Universal Robots PolyScope program: cover corner demo.urp

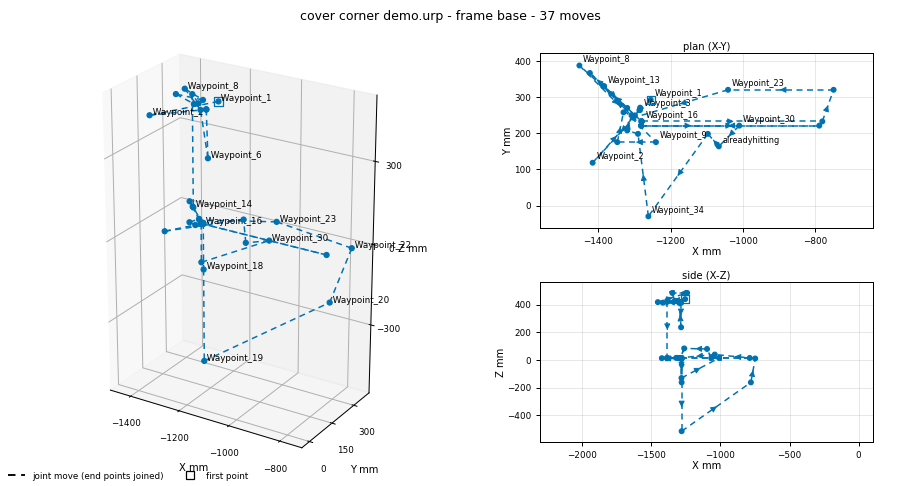
[picture p0: tool path of cover corner demo.urp in frame base, 37 of 37 moves have a stored position in this frame; points joined in program order, loops and branches not executed]
Program cover corner demo (installation=default directory=/programs createdIn=5.21.3 lastSavedIn=5.21.3 robotSerialNumber=20246801938)
Calibrated DH parameters: a=[-0.000071, -0.790281, -0.600694, 0.000061, -0.000039, 0]; d=[0.236272, 604.465945, 132.116513, -736.382239, 0.159268, 0.154005]; alpha=[1.570254, -0.000567, 0.000559, 1.571709, -1.56999, 0]; deltaTheta=[0, -0.409357, 7.293326, -0.600784, -0.000001, -0.000001]
InitVariablesNode
Robot Program (runOnlyOnce=true)
  'right cover corner weld'
  'around then straight'
  MoveJ speed 60 deg/s, acceleration 80 deg/s^2 (useActiveTCP=true optimoveEnabled=false optiMoveSpeed=0.3 optiMoveAcceleration=0.09) feature=Base
    Waypoint Waypoint_1: TCP in base x=-1254.835 y=293.144 z=440.638 mm, rx=-1.1133 ry=-2.919 rz=-0.012 rad; joints [-17.342, -68.282, 77.268, -10.218, 114.462, -0.524] deg; TCP offset x=4.51 y=-328 z=105.73 mm, rx=1.2092 ry=-1.2092 rz=1.2092 rad
  MoveJ speed 60 deg/s, acceleration 80 deg/s^2 (useActiveTCP=true optimoveEnabled=false optiMoveSpeed=0.3 optiMoveAcceleration=0.09) feature=Base
    'around'
    Waypoint Waypoint_2: TCP in base x=-1415.792 y=118.619 z=414.89 mm, rx=-1.1133 ry=-2.919 rz=-0.012 rad; joints [-6.875, -56.934, 61.751, -6.179, 124.925, -0.802] deg
    Waypoint Waypoint_3: TCP in base x=-1285.353 y=264.728 z=415.081 mm, rx=-1.1133 ry=-2.919 rz=-0.012 rad; joints [-15.395, -66.104, 76.117, -11.264, 116.409, -0.572] deg
    Waypoint Waypoint_4: TCP in base x=-1285.353 y=264.728 z=415.081 mm, rx=-0.9669 ry=-2.5613 rz=0.9063 rad; joints [-26.4, -72.021, 90.911, -20.061, 105.41, 39.121] deg
    Waypoint Waypoint_5: TCP in base x=-1285.353 y=264.728 z=415.081 mm, rx=-0.6786 ry=-1.8298 rz=1.759 rad; joints [-33.44, -66.732, 105.133, -39.549, 98.375, 88.019] deg
    Waypoint Waypoint_6: TCP in base x=-1284.072 y=271.274 z=236.976 mm, rx=-0.6786 ry=-1.8298 rz=1.759 rad; joints [-33.833, -57.911, 109.289, -52.527, 97.983, 88.015] deg
    'straight'
    Waypoint Waypoint_7: TCP in base x=-1298.614 y=249.951 z=415.063 mm, rx=1.2773 ry=-2.8625 rz=-0.028 rad; joints [-31.009, -57.342, 61.988, -4.82, 10.948, -0.916] deg
    Waypoint Waypoint_8: TCP in base x=-1452.41 y=387.964 z=419.01 mm, rx=1.2773 ry=-2.8625 rz=-0.028 rad; joints [-32.614, -38.704, 28.297, 10.236, 9.332, -0.921] deg
  'left cover corner weld'
  MoveJ speed 60 deg/s, acceleration 80 deg/s^2 (useActiveTCP=true optimoveEnabled=false optiMoveSpeed=0.3 optiMoveAcceleration=0.09) feature=Base
    Waypoint Waypoint_9: TCP in base x=-1240.368 y=175.706 z=485.383 mm, rx=-2.5614 ry=-1.6281 rz=0.6096 rad; joints [-170.603, -117.074, -63.044, -149.309, 36.236, -10.589] deg
  'involves base elbow flip'
  'cords are dangling scary close to weld tip (on robot2)'
  MoveJ speed 60 deg/s, acceleration 80 deg/s^2 (useActiveTCP=true optimoveEnabled=false optiMoveSpeed=0.3 optiMoveAcceleration=0.09) feature=Base
    Waypoint Waypoint_10: TCP in base x=-1347.448 y=175.706 z=485.383 mm, rx=-2.5106 ry=-1.5364 rz=0.247 rad; joints [-168.313, -139.19, -27.078, -189.813, 38.498, 11.145] deg
  'wrist flip. cords are away and we get more reach, but wrist flip means a close elbow'
  MoveJ speed 60 deg/s, acceleration 80 deg/s^2 (useActiveTCP=true optimoveEnabled=false optiMoveSpeed=0.3 optiMoveAcceleration=0.09) feature=Base
    Waypoint Waypoint_11: TCP in base x=-1330.269 y=258.318 z=427.852 mm, rx=-2.7288 ry=-1.2659 rz=-0.0761 rad; joints [-172.786, -148.887, -40.082, 1.273, -47.983, 190.799] deg
    Waypoint Waypoint_12: TCP in base x=-1319.93 y=270.458 z=428.193 mm, rx=-2.8543 ry=-1.2377 rz=-0.0137 rad; joints [-174.9, -150.783, -34.37, 3.734, -48.225, 182.288] deg
    Waypoint Waypoint_13: TCP in base x=-1383.928 y=330.345 z=430.336 mm, rx=-2.8543 ry=-1.2377 rz=-0.0137 rad; joints [-177.317, -163.409, -7.801, -10.266, -45.796, 182.378] deg
  'lift column raise. raised to be even with cover (400mm)'
  MoveJ speed 60 deg/s, acceleration 80 deg/s^2 (useActiveTCP=true optimoveEnabled=false optiMoveSpeed=0.3 optiMoveAcceleration=0.09) feature=Base
    Waypoint Waypoint_14: TCP in base x=-1383.928 y=330.345 z=12.421 mm, rx=-2.8543 ry=-1.2377 rz=-0.0137 rad; joints [-177.314, -169.954, -26.885, 15.371, -45.807, 182.367] deg
    Waypoint Waypoint_15: TCP in base x=-1423.443 y=367.323 z=13.744 mm, rx=-2.8543 ry=-1.2377 rz=-0.0137 rad; joints [-178.706, -181.113, -2.242, 1.851, -44.403, 182.419] deg
    'above point is as far back as robot can reach (7 inches when box is centered and at near side of green tape)'
    Waypoint Waypoint_16: TCP in base x=-1280.044 y=233.133 z=8.941 mm, rx=-2.8543 ry=-1.2377 rz=-0.0137 rad; joints [-173.278, -159.438, -50.801, 28.856, -49.855, 182.23] deg
    Waypoint Waypoint_21: TCP in base x=-1280.044 y=233.133 z=13.157 mm, rx=-2.1144 ry=-0.9283 rz=0.4027 rad; joints [-165.117, -154.877, -73.484, 47.103, -58.025, 230.171] deg
    Waypoint Waypoint_17: TCP in base x=-1280.044 y=233.133 z=13.157 mm, rx=-1.4551 ry=-0.6485 rz=0.6266 rad; joints [-162.22, -164.866, -73.666, 57.306, -60.921, 271.226] deg
    Waypoint Waypoint_18: TCP in base x=-1280.044 y=233.133 z=-161.418 mm, rx=-1.4551 ry=-0.6485 rz=0.6266 rad; joints [-162.214, -175.589, -65.432, 59.795, -60.923, 271.225] deg
    'plenty of space to godown hella far. about 2.5 feet'
    Waypoint Waypoint_19: TCP in base x=-1280.044 y=233.133 z=-514.411 mm, rx=-1.4551 ry=-0.6485 rz=0.6266 rad; joints [-162.197, -202.133, -33.245, 54.157, -60.925, 271.214] deg
    'plenty of space to go in farther. about 1.5 feet'
    Waypoint Waypoint_20: TCP in base x=-779.391 y=233.133 z=-161.418 mm, rx=-1.4551 ry=-0.6485 rz=0.6266 rad; joints [-150.184, -170.388, -110.718, 99.965, -72.968, 270.973] deg
    'the entire path can be a lot closer. at least a foot closer'
    'backaway:'
    Waypoint Waypoint_22: TCP in base x=-748.166 y=320.706 z=11.481 mm, rx=-2.7733 ry=1.3401 rz=-0.0046 rad; joints [-197.66, -122.46, -96.634, -139.289, -236.108, 4.164] deg
    Waypoint Waypoint_23: TCP in base x=-1040.583 y=320.706 z=40.127 mm, rx=-2.8835 ry=1.0826 rz=0.004 rad; joints [-191.99, -137.934, -64.751, -155.778, -240.879, 4.016] deg
    'above waypoint collides: back of welder hits cordage on forearm'
  'undo wrist flip with column raise'
  MoveJ speed 60 deg/s, acceleration 80 deg/s^2 (useActiveTCP=true optimoveEnabled=false optiMoveSpeed=0.3 optiMoveAcceleration=0.09) feature=Base
    Waypoint Waypoint_24: TCP in base x=-1302.623 y=243.502 z=15.13 mm, rx=-2.912 ry=-1.1752 rz=-0.0069 rad; joints [-174.548, -152.125, -38.795, -169.497, 51.485, 0.259] deg
    Waypoint Waypoint_25: TCP in base x=-1387.012 y=331.02 z=15.089 mm, rx=-2.912 ry=-1.1752 rz=-0.0069 rad; joints [-178.035, -170.27, -0.309, -189.867, 47.978, 0.301] deg
    Waypoint Waypoint_26: TCP in base x=-1281.32 y=221.409 z=15.14 mm, rx=-2.912 ry=-1.1752 rz=-0.0069 rad; joints [-173.603, -149.923, -43.327, -167.161, 52.432, 0.25] deg
    Waypoint Waypoint_27: TCP in base x=-1281.32 y=221.409 z=15.14 mm, rx=-2.3478 ry=-0.9496 rz=0.3068 rad; joints [-166.978, -141.646, -65.889, -152.84, 59.069, 36.679] deg
    Waypoint turnwayinside: TCP in base x=-787.829 y=221.409 z=15.14 mm, rx=-2.3478 ry=-0.9496 rz=0.3068 rad; joints [-159.32, -115.922, -116.47, -127.953, 66.754, 36.618] deg
    Waypoint Waypoint_28: TCP in base x=-1281.32 y=221.409 z=15.14 mm, rx=-1.4895 ry=-0.6052 rz=0.5951 rad; joints [-161.902, -148.139, -77.504, -134.714, 64.152, 89.869] deg
    Waypoint Waypoint_29: TCP in base x=-1281.32 y=221.409 z=-129.88 mm, rx=-1.4895 ry=-0.6052 rz=0.5951 rad; joints [-161.898, -155.56, -75.62, -129.177, 64.155, 89.87] deg
    'bavkaway'
    Waypoint Waypoint_30: TCP in base x=-1009.408 y=221.409 z=15.14 mm, rx=2.9043 ry=-1.1922 rz=0.0065 rad; joints [-189.438, -134.893, -73.428, -152.046, 125.205, -0.215] deg
    Waypoint alreadyhitting: TCP in base x=-1066.118 y=163.974 z=15.167 mm, rx=2.9043 ry=-1.1922 rz=0.0065 rad; joints [-186.508, -137.271, -68.77, -154.339, 128.132, -0.238] deg
  'backaway 2'
  MoveJ speed 60 deg/s, acceleration 80 deg/s^2 (useActiveTCP=true optimoveEnabled=false optiMoveSpeed=0.3 optiMoveAcceleration=0.09) feature=Base
    Waypoint Waypoint_31: TCP in base x=-1096.486 y=198.657 z=80.338 mm, rx=2.9721 ry=-0.9596 rz=0.0188 rad; joints [-23.586, -40.373, 58.89, -17.461, -77.751, -1.037] deg
    Waypoint Waypoint_34: TCP in base x=-1261.306 y=-29.905 z=84.211 mm, rx=2.9721 ry=-0.9596 rz=0.0188 rad; joints [-12.627, -29.552, 36.988, -6.309, -66.8, -1.255] deg
    Waypoint farthestitgoes: TCP in base x=-1290.074 y=198.657 z=15.949 mm, rx=2.9721 ry=-0.9596 rz=0.0188 rad; joints [-20.678, -20.111, 22.774, -1.594, -74.856, -1.089] deg
    Waypoint Waypoint_32: TCP in base x=-1319.947 y=208.204 z=15.949 mm, rx=2.9721 ry=-0.9596 rz=0.0188 rad; joints [-20.614, -9.578, 0.171, 10.477, -74.803, -1.09] deg
    Waypoint Waypoint_33: TCP in base x=-1308.108 y=249.99 z=15.949 mm, rx=2.9721 ry=-0.9596 rz=0.0188 rad; joints [-22.198, -11.648, 4.673, 8.037, -76.385, -1.06] deg
